(* CODESYS project SHSNU_monitor.project

Project tree, tasks and I/O mapping:
  Device : OWEN PLC323.03-CS.WEB, Owen, order no. 005, version 3.5.0.40
      unmapped channels: Discrete Outputs, Discrete inputs
    application Application
      libraries: CoDeSys Container Library Template, 3.5.3.0 (3S - Smart Software Solutions GmbH); МВА АСКИР, 1.0.0.0 (ООО ПЛАДА); ModBus, 3.1.1 (OWEN); SysCom, 3.5.5.0 (System); ModulsOwenLib, 3.5.4.2 (Production association OWEN); OwenArchiverErrors, 3.5.4.2 (Production association OWEN); CAA Async Manager Extern, * (CAA Technical Workgroup); ArchivatorOwenLib, 3.5.4.2 (OWEN); SysTime23, 3.5.2.0 (System); SysTimeRtc, 3.5.5.0 (System); CAA DTUtil Extern, * (CAA Technical Workgroup); CAA File, 3.5.11.0 (CAA Technical Workgroup); SysSocket, 3.5.9.0 (System); OwenModemLib, 3.5.2.13 (OWEN); BASIC, 3.31 (OSCAT)
      task MainTask (cyclic, interval t#20ms, priority 1, watchdog t#5000ms x 1) calls PLC_PRG
      program PLC_PRG [CFC]
      Symbols
      global variables GVL
      data type Massive
      Code/
        Dop_modules/
          program convert [ST]
          function Duo_Word_to_Real [CFC]
          function block Real_to_Duo_Word [CFC]
          function block Perecl_Perem [ST]
          function block Timer_impuls [CFC]
          function block Schetchik [ST]
          function block NotNull [ST]
          function block IVD3_input_old [ST]
          function block IVD3_input_reg [ST]
          function POU [CFC]
          function block AddInMassive [ST]
          function block IVD3_input [ST]
          function block Auton_val [ST]
        Modules/
          function block DTime [ST]
          function block SPLIT_DT_TO_FSTRINGS [ST]
          function CONCAT11 [ST]
          function LEAD_ZERO [ST]
          function block SMS [CFC]
        Modules_dinamogramma/
          function block MassivCollect [ST]
          function block Create_Shablon [ST]
          function block Alarm_Control [ST]
          function block Correct_Shablon [ST]
          function block Auton_dynamogram_modbus [ST]
          function block Create_Shablon_v2 [ST]
        Modules_parameter/
          function block Calculate_Parameter_Usilie [ST]
          function block Emulate_Parameter_Power [ST]
      data type AlarmLog
    Ethernet : Ethernet, 3S - Smart Software Solutions GmbH, version 3.4.2.0
      ModbusTCP_Slave_Device : ModbusTCP Slave Device, 3S - Smart Software Solutions GmbH, version 3.4.1.10
          settings: Unit-ID = 159
          input  p13 : WORD  // IW0
          input  p14 : WORD  // IW1
          input  p15 : WORD  // IW2
          input  p16 : WORD  // IW3
          input  p17 : WORD  // IW4
          input  p18 : WORD  // IW5
          input  p19 : WORD  // IW6
          input  p20 : WORD  // IW7
          input  p21 : WORD  // IW8
          input  p22 : WORD  // IW9
          unmapped channels: QW0, QW1, QW2, QW3, QW4, QW5, QW6, QW7, QW8, QW9
    Owen:Internal
        output Application.ledError : BOOL  // Discrete Outputs.RELE1
        output Application.ledError : BOOL  // Discrete Outputs.LED_ERROR
        unmapped channels: Discrete Outputs, Discrete inputs
  text list GlobalTextList
  5ce3da45-db07-42e7-a21c-a00fff4ed8f6|D:\Work\Gorizont REP\code\src\Askir\DesktopApp\res\dashboard.jpg
  5ce3da45-db07-42e7-a21c-a00fff4ed8f6|F:\Other\YandexDisk\OVEN\Документация\dashboard.jpg
  5ce3da45-db07-42e7-a21c-a00fff4ed8f6|F:\Other\YandexDisk\OVEN\Проекты\Askir\Askir_materials\Askir_bg.jpg
  5ce3da45-db07-42e7-a21c-a00fff4ed8f6|F:\Other\YandexDisk\OVEN\Проекты\Askir\Askir_materials\ZadPodElDv.jpg
  5ce3da45-db07-42e7-a21c-a00fff4ed8f6|F:\Other\YandexDisk\OVEN\Проекты\Askir\Askir_materials\Askir_bg_lable.jpg
*)

// Device/Application/Massive
TYPE Massive :
STRUCT
	Date_Time: STRING(20);
	var1, var2, var3, var4, var5, var6 : REAL;
END_STRUCT
END_TYPE

// Device/Application/AlarmLog
TYPE AlarmLog :
STRUCT
	Date_Time: STRING(20);
	ShablonIndex:INT;
	ShablonValue:REAL;
	Value:REAL;
	Otklonenie:REAL;
END_STRUCT
END_TYPE

// Device/Application/GVL
VAR_GLOBAL
	var2: REAL;
	
	p1, p2, p3, p4, p5, p6, p7, p8, p9, p10: WORD;
	
	
	VibrA1, VibrA2, VibrA3, VibrB1, VibrB2, VibrB3, VibrC1, VibrC2, VibrC3, VibrD1, VibrD2, VibrD3: REAL;
	(*Вибрация позиция A плоскость X*)		VibrAX:REAL;
	(*Вибрация позиция A плоскость Y*)		VibrAY:REAL;
	(*Вибрация позиция A плоскость Z*)		VibrAZ:REAL;
	
	(*Вибрация позиция B плоскость X*)		VibrBX:REAL;
	(*Вибрация позиция B плоскость Y*)		VibrBY:REAL;
	(*Вибрация позиция B плоскость Z*)		VibrBZ:REAL;
	
	(*Вибрация позиция C плоскость X*)		VibrCX:REAL;
	(*Вибрация позиция C плоскость Y*)		VibrCY:REAL;
	(*Вибрация позиция C плоскость Z*)		VibrCZ:REAL;
	
	(*Динамограмма с датчика усилия*)		Dinamogram: ARRAY[1..Dynamogram_length] OF INT;
	minMnoj: REAL := 0.001;
	maxMnoj: REAL := 100;
	
	minSmesh: REAL := -100;
	maxSmesh: REAL := 100;
	
	Start: BOOL := FALSE;
	
	arrey1111 : ARRAY [1..5] OF INT := [1 , 2, 3, 4, 5];
	ledError: BOOL:=TRUE;
	
	
END_VAR

VAR_GLOBAL RETAIN
	M1, M2, M3, M4, M5, M6, M7, M8, M9, M10, M11, M12: REAL := 1;
	S1, S2, S3, S4, S5, S6, S7, S8, S9, S10, S11, S12: REAL := 0;
	MemM1, MemM2, MemM3, MemM4, MemM5, MemM6, MemM7, MemM8, MemM9, MemM10, MemM11, MemM12: REAL;
	MemS1, MemS2, MemS3, MemS4, MemS5, MemS6, MemS7, MemS8, MemS9, MemS10, MemS11, MemS12: REAL;
	SaveConfig: BOOL;
	
END_VAR

VAR_GLOBAL CONSTANT
	m_MAX_arr: INT:=500; //размер массива	
	Dynamogram_length: INT:=500;
END_VAR

// Device/Application/PLC_PRG
PROGRAM PLC_PRG
VAR
	tp1: TP;
	ErrMDVV: WORD;
	v4: REAL;
	v3: REAL;
	v2: REAL;
	v1: REAL;
	x: BYTE;
	R1, R2, R3, R4, R5, R6, R7, R8, R9, R10, R11, R12, R13, R14, R15, R16, R17, R18, R19, R20, R21, R22: REAL;
	peremR: REAL;
	x3: WORD;
	Perecluchatel: Perecl_Perem;
	RS_0: RS;
	v1_2: REAL;
	v1_3: REAL;
	v2_2: REAL;
	v3_2: REAL;
	v4_2: REAL;
	v1_2IS: WORD;
	v2_2IS: WORD;
	v3_2IS: WORD;
	v4_2IS: WORD;
	v5_2: REAL;
	v6_2: REAL;
	v7_2: REAL;
	v5_2IS: WORD;
	v6_2IS: WORD;
	v7_2IS: WORD;
	v8_2: REAL;
	cicle: WORD;
	Sch_1: Schetchik;
	
	NotNull_1: NotNull;
	NotNull_2: NotNull;
	NotNull_3: NotNull;
	NotNull_4: NotNull;
	NotNull_5: NotNull;
	NotNull_6: NotNull;
	NotNull_7: NotNull;
	NotNull_8: NotNull;
	NotNull_9: NotNull;
	NotNull_10: NotNull;
	
	MConf1,MConf2,MConf3,MConf4,MConf5,MConf6,MConf7,MConf8,MConf9,MConf10,MConf11,MConf12, MConfigTest:REAL := 1;
	SConf1,SConf2,SConf3,SConf4,SConf5,SConf6,SConf7,SConf8,SConf9,SConf10,SConf11,SConf12, SConfigTest:REAL := 1;
	
	
	//IVD3_input_reg_0: IVD3_input_reg;
	//IVD3_input_reg_1: IVD3_input_reg;
	//IVD3_input_reg_2: IVD3_input_reg;
	//IVD3_input_reg_3: IVD3_input_reg;
	
	Port_5: ComConn;
	MV110_8A: MV110_8A_inputs;
	
	MV110_8A_inp_1,
	MV110_8A_inp_2, 
	MV110_8A_inp_3, 
	MV110_8A_inp_4, 
	MV110_8A_inp_5, 
	MV110_8A_inp_6, 
	MV110_8A_inp_7, 
	MV110_8A_inp_8: REAL;
	
	ComConn_Tablo: ComConn;
	Write_in_Tablo: UniWrite;
	ComConn_Vibro: ComConn;
	SR_0: RS;
	

	


	DTime_0: DTime;
	
	systimestring:string;
	vcb: DWORD;

	
	testMassiv: Massive := (Date_Time:= systimestring, var1:=VibrAZ, var2:=VibrAX, var3:=VibrAY, var4:=VibrBZ, var5:=VibrBX, var6:=VibrBY);
	AddInMassive_0: AddInMassive;
	
	
	MassivIVD3_1, MassivIVD3_2, MassivIVD3_3: ARRAY [0..gvl.m_MAX_arr] OF REAL;
	timeMassiveIVD3_1, timeMassiveIVD3_2, timeMassiveIVD3_3: STRING;
	
	TP_add_massiv: TP;
	RS_TP: RS;
	Emulate_Parameter_Power_test: Emulate_Parameter_Power;
	
	Power_U: REAL;
	Power_I: REAL;
	Power_Work_Hod:REAL;
	Power_Work_Up:REAL;
	Power_Work_Down:REAL;
	Power_Min:REAL;
	Power_Max:REAL;
	Power_Razmah:REAL;
	
	Calculate_Parameter_Usilie_0: Calculate_Parameter_Usilie;
	
	Usilie_Work_Hod:REAL;
	Usilie_Work_Up:REAL;
	Usilie_Work_Down:REAL;
	Usilie_Raznica:REAL;
	Usilie_Min:REAL;
	Usilie_Max:REAL;
	Usilie_Razmah:REAL;
	ComConn_Sim: comconn;
	modem_fb: FB_SMS_CSD;
	
	newSMS, newRing, CSD, modem_busy: BOOL;
	
	tesTP: bool;
	TON_0, TON_1, TON_2: ton;
	start: bool := true;
	R_TRIG_0: R_TRIG;
	F_TRIG_0: F_TRIG;
	TON_3: ton;
	RS_1: rs;
	qwe: IVD3_input_reg;
	asd: IVD3_input_reg;
	zxc: IVD3_input_reg;
	IVD3_input_reg_0: IVD3_input_reg;
	Auton_val_0: Auton_val;
	auton_value: INT;
	MassivCollect_Dynamogram: MassivCollect;
	masDynamogram: ARRAY [0..gvl.m_MAX_arr] OF REAL;
	timeDynamogram: STRING;
	auton_val_time: STRING;
	TP_work: TP;
	Start_work: BOOL:= false;
	IVD3_A: IVD3_input_reg;
	IVD3_B: IVD3_input_reg;
	IVD3_C: IVD3_input_reg;
END_VAR
VAR // added by the converter: edge detectors and wires of the graphical bodies
    _w1 : BYTE;
END_VAR

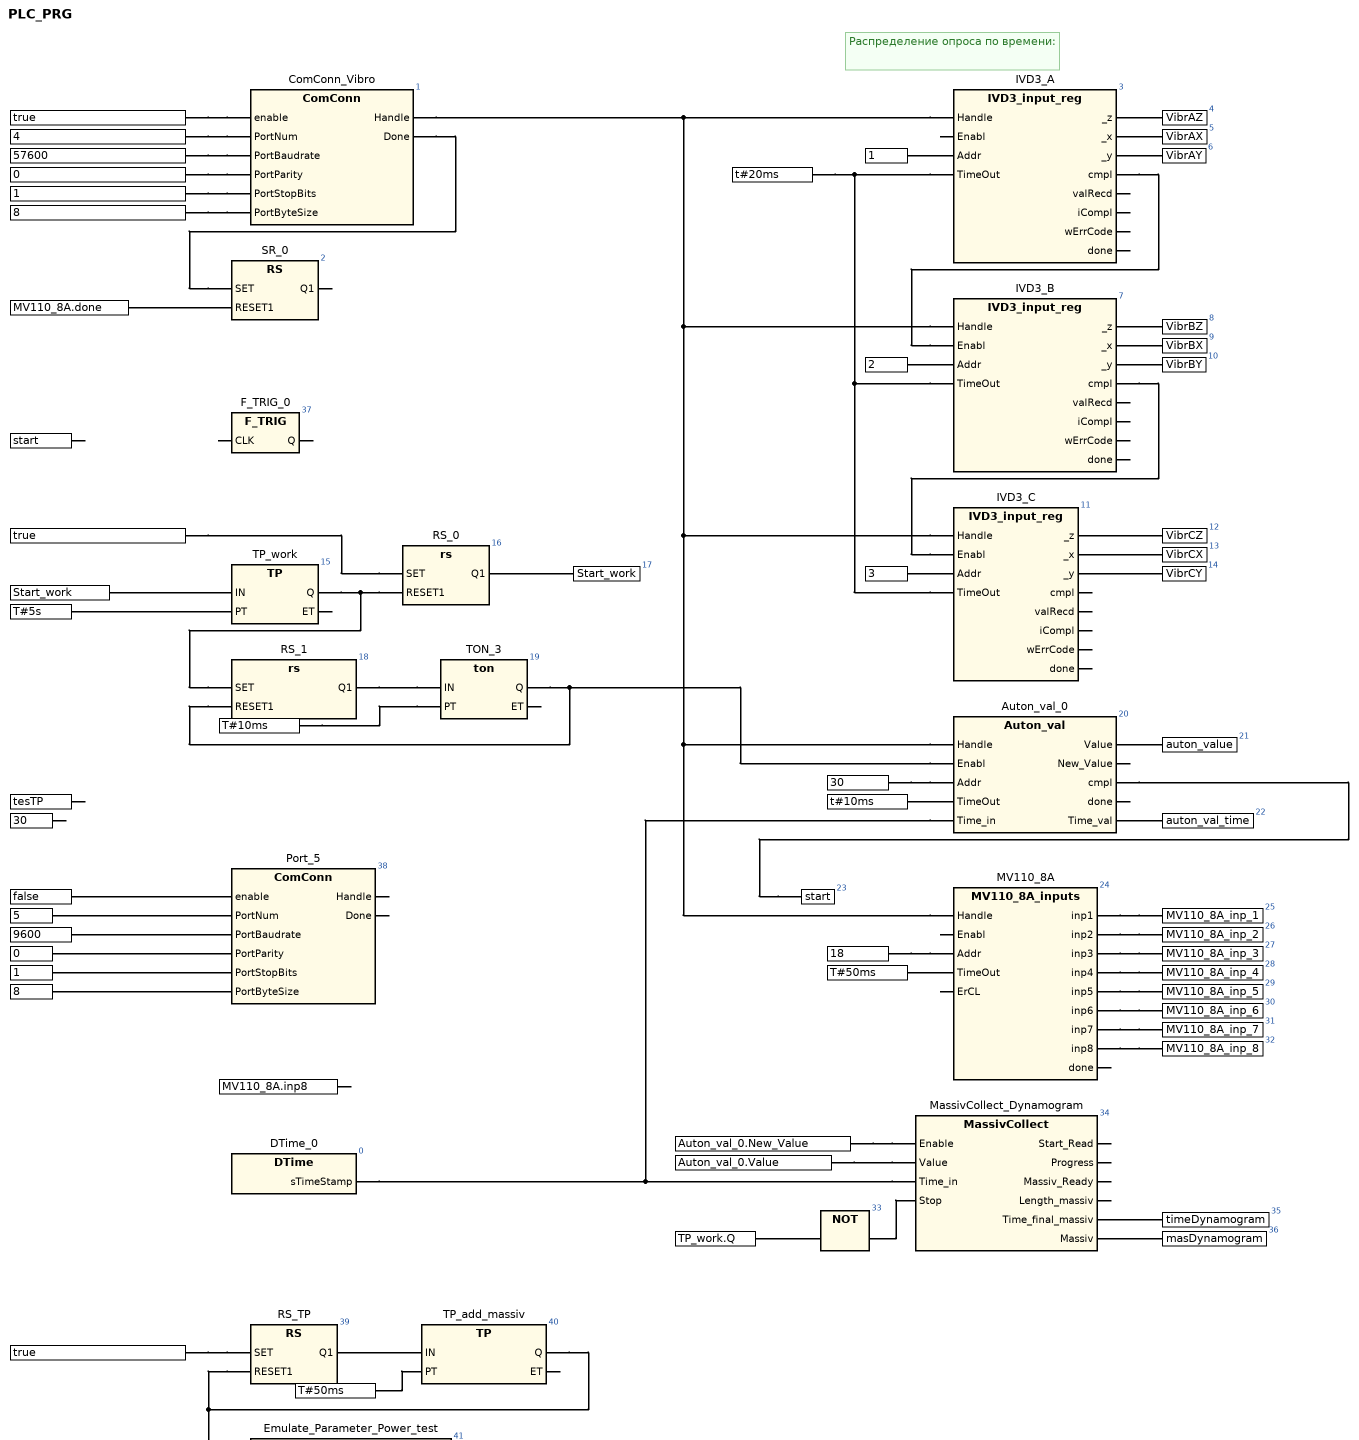
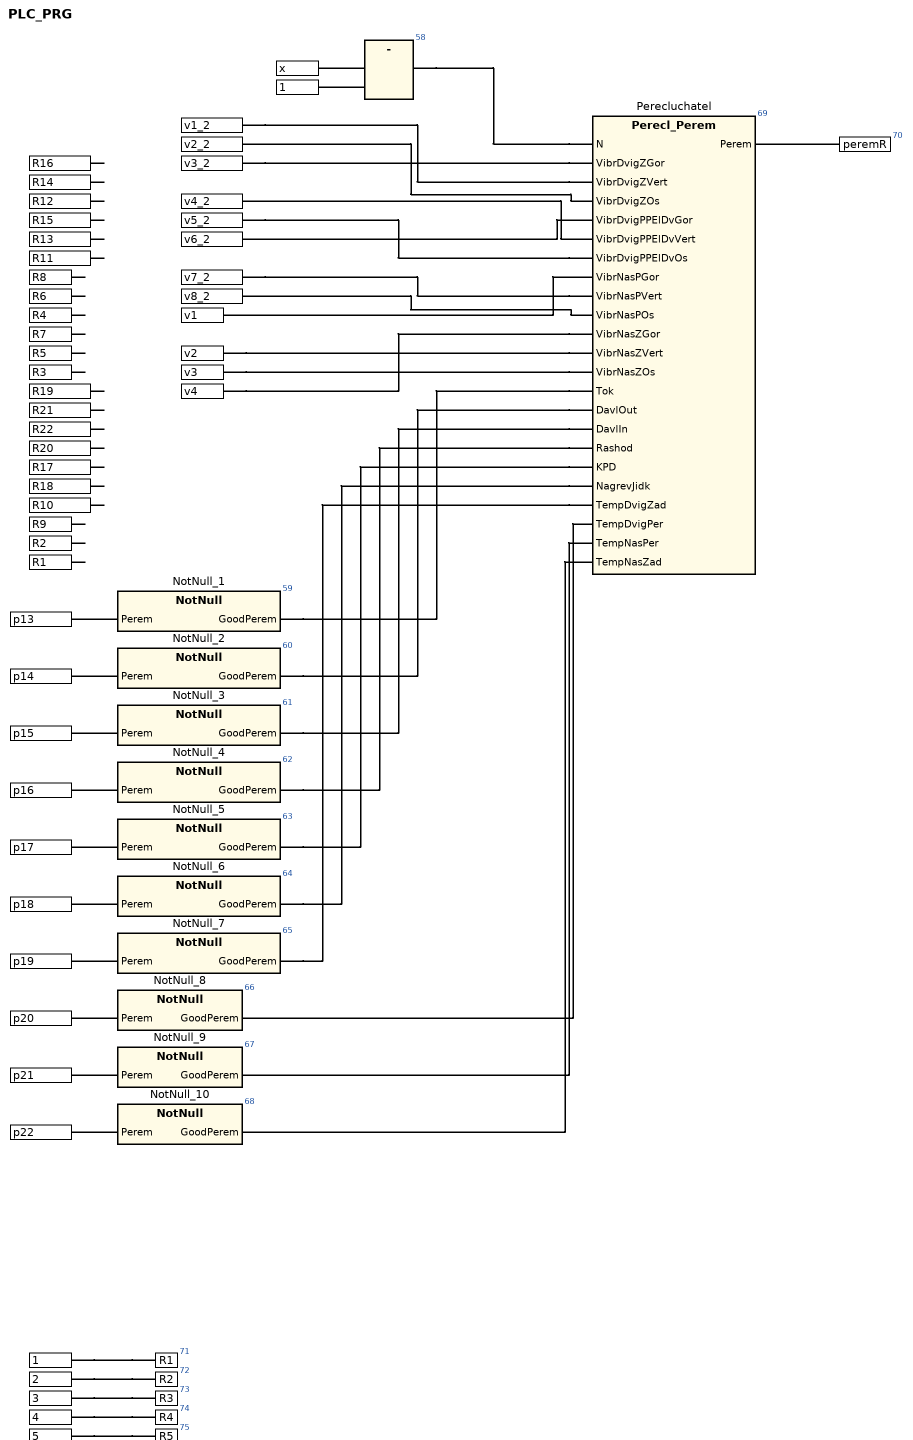
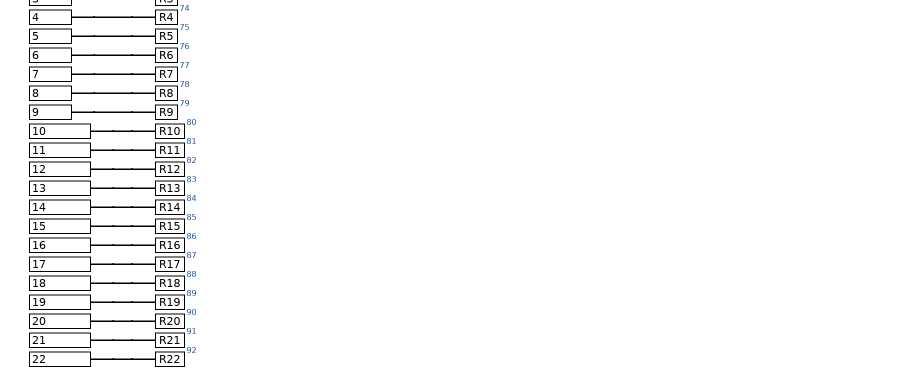
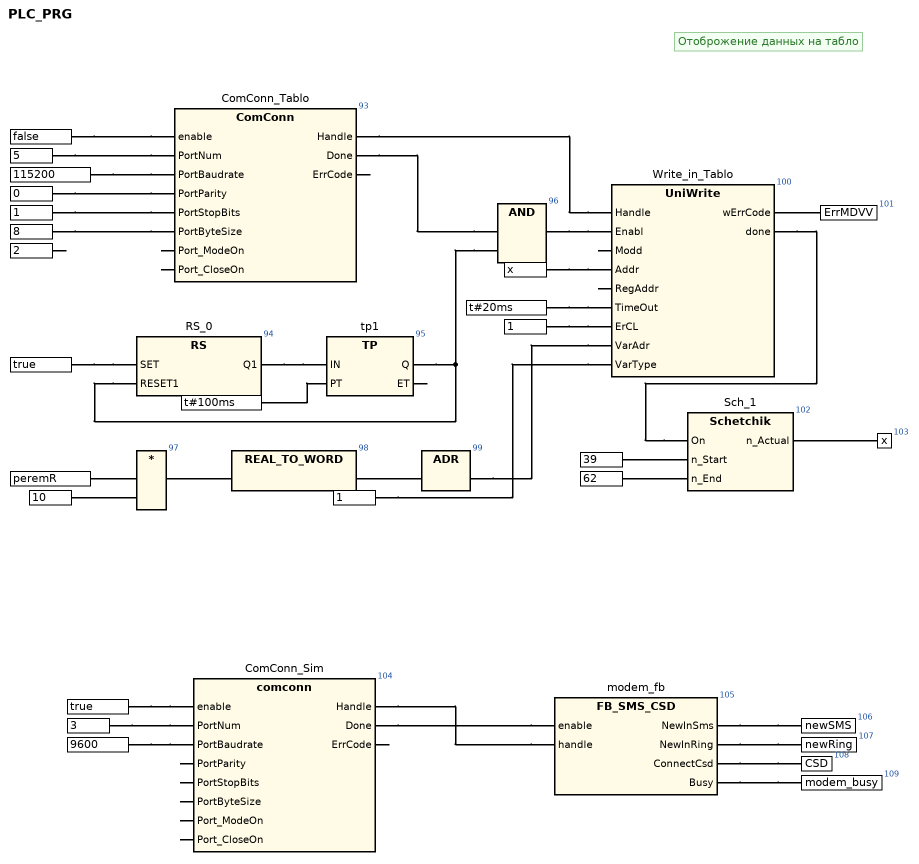
DTime_0(); // DTime
ComConn_Vibro(
    enable := true,
    PortNum := 4,
    PortBaudrate := 57600,
    PortParity := 0,
    PortStopBits := 1,
    PortByteSize := 8); // ComConn
SR_0(SET := ComConn_Vibro.Done, RESET1 := MV110_8A.done); // RS
// Распределение опроса по времени:
IVD3_A(Handle := ComConn_Vibro.Handle, Addr := 1, TimeOut := t#20ms); // IVD3_input_reg
VibrAZ := IVD3_A._z;
VibrAX := IVD3_A._x;
VibrAY := IVD3_A._y;
IVD3_B(Handle := ComConn_Vibro.Handle, Enabl := IVD3_A.cmpl, Addr := 2, TimeOut := t#20ms); // IVD3_input_reg
VibrBZ := IVD3_B._z;
VibrBX := IVD3_B._x;
VibrBY := IVD3_B._y;
IVD3_C(Handle := ComConn_Vibro.Handle, Enabl := IVD3_B.cmpl, Addr := 3, TimeOut := t#20ms); // IVD3_input_reg
VibrCZ := IVD3_C._z;
VibrCX := IVD3_C._x;
VibrCY := IVD3_C._y;
TP_work(IN := Start_work, PT := T#5s); // TP
RS_0(SET := true, RESET1 := TP_work.Q); // rs
Start_work := RS_0.Q1;
RS_1(SET := TP_work.Q, RESET1 := TON_3.Q); // rs
TON_3(IN := RS_1.Q1, PT := T#10ms); // ton
Auton_val_0(
    Handle := ComConn_Vibro.Handle,
    Enabl := TON_3.Q,
    Addr := 30,
    TimeOut := t#10ms,
    Time_in := DTime_0.sTimeStamp); // Auton_val
auton_value := Auton_val_0.Value;
auton_val_time := Auton_val_0.Time_val;
start := Auton_val_0.cmpl;
MV110_8A(Handle := ComConn_Vibro.Handle, Addr := 18, TimeOut := T#50ms); // MV110_8A_inputs
MV110_8A_inp_1 := MV110_8A.inp1;
MV110_8A_inp_2 := MV110_8A.inp2;
MV110_8A_inp_3 := MV110_8A.inp3;
MV110_8A_inp_4 := MV110_8A.inp4;
MV110_8A_inp_5 := MV110_8A.inp5;
MV110_8A_inp_6 := MV110_8A.inp6;
MV110_8A_inp_7 := MV110_8A.inp7;
MV110_8A_inp_8 := MV110_8A.inp8;
MassivCollect_Dynamogram(
    Enable := Auton_val_0.New_Value,
    Value := Auton_val_0.Value,
    Time_in := DTime_0.sTimeStamp,
    Stop := NOT TP_work.Q); // MassivCollect
timeDynamogram := MassivCollect_Dynamogram.Time_final_massiv;
masDynamogram := MassivCollect_Dynamogram.Massiv;
F_TRIG_0(); // F_TRIG
Port_5(
    enable := false,
    PortNum := 5,
    PortBaudrate := 9600,
    PortParity := 0,
    PortStopBits := 1,
    PortByteSize := 8); // ComConn
RS_TP(SET := true, RESET1 := TP_add_massiv.Q); // RS
TP_add_massiv(IN := RS_TP.Q1, PT := T#50ms); // TP
Emulate_Parameter_Power_test(
    Enable := TP_add_massiv.Q,
    U_Random_Min := 370,
    U_Random_Max := 390,
    I_Random_Min := 40,
    I_Random_Max := 60,
    Index := MassivCollect_Dynamogram.Progress); // Emulate_Parameter_Power
Power_U := Emulate_Parameter_Power_test.U;
Power_I := Emulate_Parameter_Power_test.I;
Power_Work_Up := Emulate_Parameter_Power_test.Work_Up;
Power_Work_Down := Emulate_Parameter_Power_test.Work_Down;
Power_Work_Hod := Emulate_Parameter_Power_test.Work_Hod;
Power_Max := Emulate_Parameter_Power_test.Max_Power;
Power_Min := Emulate_Parameter_Power_test.Min_Power;
Power_Razmah := Emulate_Parameter_Power_test.Razmah;
Calculate_Parameter_Usilie_0(
    Enable := MassivCollect_Dynamogram.Massiv_Ready,
    Index := MassivCollect_Dynamogram.Progress,
    Dinamogramma := MassivCollect_Dynamogram.Massiv); // Calculate_Parameter_Usilie
Usilie_Work_Up := Calculate_Parameter_Usilie_0.Work_Up;
Usilie_Work_Down := Calculate_Parameter_Usilie_0.Work_Down;
Usilie_Work_Hod := Calculate_Parameter_Usilie_0.Work_Hod;
Usilie_Raznica := Calculate_Parameter_Usilie_0.Raznica;
Usilie_Max := Calculate_Parameter_Usilie_0.Max_Usil;
Usilie_Min := Calculate_Parameter_Usilie_0.Min_Usil;
Usilie_Razmah := Calculate_Parameter_Usilie_0.Razmah;
_w1 := x - 1;
NotNull_1(Perem := p13); // NotNull
NotNull_2(Perem := p14); // NotNull
NotNull_3(Perem := p15); // NotNull
NotNull_4(Perem := p16); // NotNull
NotNull_5(Perem := p17); // NotNull
NotNull_6(Perem := p18); // NotNull
NotNull_7(Perem := p19); // NotNull
NotNull_8(Perem := p20); // NotNull
NotNull_9(Perem := p21); // NotNull
NotNull_10(Perem := p22); // NotNull
Perecluchatel(
    N := _w1,
    VibrDvigZGor := v3_2,
    VibrDvigZVert := v1_2,
    VibrDvigZOs := v2_2,
    VibrDvigPPElDvGor := v6_2,
    VibrDvigPPElDvVert := v4_2,
    VibrDvigPPElDvOs := v5_2,
    VibrNasPGor := v1,
    VibrNasPVert := v7_2,
    VibrNasPOs := v8_2,
    VibrNasZGor := v4,
    VibrNasZVert := v2,
    VibrNasZOs := v3,
    Tok := NotNull_1.GoodPerem,
    DavlOut := NotNull_2.GoodPerem,
    DavlIn := NotNull_3.GoodPerem,
    Rashod := NotNull_4.GoodPerem,
    KPD := NotNull_5.GoodPerem,
    NagrevJidk := NotNull_6.GoodPerem,
    TempDvigZad := NotNull_7.GoodPerem,
    TempDvigPer := NotNull_8.GoodPerem,
    TempNasPer := NotNull_9.GoodPerem,
    TempNasZad := NotNull_10.GoodPerem); // Perecl_Perem
peremR := Perecluchatel.Perem;
R1 := 1;
R2 := 2;
R3 := 3;
R4 := 4;
R5 := 5;
R6 := 6;
R7 := 7;
R8 := 8;
R9 := 9;
R10 := 10;
R11 := 11;
R12 := 12;
R13 := 13;
R14 := 14;
R15 := 15;
R16 := 16;
R17 := 17;
R18 := 18;
R19 := 19;
R20 := 20;
R21 := 21;
R22 := 22;
ComConn_Tablo(
    enable := false,
    PortNum := 5,
    PortBaudrate := 115200,
    PortParity := 0,
    PortStopBits := 1,
    PortByteSize := 8); // ComConn
RS_0(SET := true, RESET1 := tp1.Q); // RS
tp1(IN := RS_0.Q1, PT := t#100ms); // TP
// Отоброжение данных на табло
Write_in_Tablo(
    Handle := ComConn_Tablo.Handle,
    Enabl := ComConn_Tablo.Done AND tp1.Q,
    Addr := x,
    TimeOut := t#20ms,
    ErCL := 1,
    VarAdr := ADR(REAL_TO_WORD(peremR * 10)),
    VarType := 1); // UniWrite
ErrMDVV := Write_in_Tablo.wErrCode;
Sch_1(On := Write_in_Tablo.done, n_Start := 39, n_End := 62); // Schetchik
x := Sch_1.n_Actual;
ComConn_Sim(enable := true, PortNum := 3, PortBaudrate := 9600); // comconn
modem_fb(enable := ComConn_Sim.Done, handle := ComConn_Sim.Handle); // FB_SMS_CSD
newSMS := modem_fb.NewInSms;
newRing := modem_fb.NewInRing;
CSD := modem_fb.ConnectCsd;
modem_busy := modem_fb.Busy;
// start: input not connected
// tesTP: input not connected
// 30: input not connected
// MV110_8A.inp8: input not connected
// MassivCollect_Dynamogram.Length_massiv: input not connected
// R16: input not connected
// R14: input not connected
// R12: input not connected
// R15: input not connected
// R13: input not connected
// R11: input not connected
// R8: input not connected
// R6: input not connected
// R4: input not connected
// R7: input not connected
// R5: input not connected
// R3: input not connected
// R19: input not connected
// R21: input not connected
// R22: input not connected
// R20: input not connected
// R17: input not connected
// R18: input not connected
// R10: input not connected
// R9: input not connected
// R2: input not connected
// R1: input not connected
// 2: input not connected

END_PROGRAM

// Device/Application/Code/Modules/DTime
FUNCTION_BLOCK DTime
VAR_OUTPUT
	sTimeStamp:						STRING(20);							// метка времени в виде форматированной строки
END_VAR
VAR
	fbGetCurrentDT:					DTU.GetDateAndTime;					// ФБ считывания системного времени	
	fbSplitDT:						SPLIT_DT_TO_FSTRINGS;				// ФБ конвертации времени в строку
	asDateTimeStrings:				ARRAY [0..10] OF STRING;			// метка времени в виде отдельных строковых разрядов
	
END_VAR
VAR CONSTANT
	// заголовок архива
	c_sTitle:						STRING(60)	:=	'Дата;Время;Значение типа WORD;Значение типа REAL;$N';
	c_sDelimiter:					STRING(1)	:=	';';
END_VAR

// считываем системное время
fbGetCurrentDT(xExecute:=NOT(fbGetCurrentDT.xDone));

IF fbGetCurrentDT.xDone THEN
	// вырезаем отдельные разряды времени и конвертируем их в строки
	fbSplitDT(dtDateAndTime:=fbGetCurrentDT.dtDateAndTime);
END_IF

// подготавливаем метку времени в виде форматированной строки
asDateTimeStrings[0]	:=	fbSplitDT.sDay;
asDateTimeStrings[1]	:=	'.';
asDateTimeStrings[2]	:=	fbSplitDT.sMonth;
asDateTimeStrings[3]	:=	'.';
asDateTimeStrings[4]	:=	fbSplitDT.sYear;
asDateTimeStrings[5]	:=	c_sDelimiter;
asDateTimeStrings[6]	:=	fbSplitDT.sHour;
asDateTimeStrings[7]	:=	':';
asDateTimeStrings[8]	:=	fbSplitDT.sMinute;
asDateTimeStrings[9]	:=	':';
asDateTimeStrings[10]	:=	fbSplitDT.sSecond;

// собираем дату и время в строку
sTimeStamp:= CONCAT11(asDateTimeStrings);

END_FUNCTION_BLOCK

// Device/Application/Code/Modules/CONCAT11
// функция склеивает заданное число строковых переменных, помещенных в массив

FUNCTION CONCAT11 : STRING(255)
VAR_INPUT
	asSTR:			ARRAY [0..c_MAX_STR] OF STRING;
END_VAR
VAR
	sBuffer:		STRING;			// промежуточная переменная
	i:				INT;			// счетчик для цикла
END_VAR

VAR CONSTANT
	c_MAX_STR:		INT:=10;		// размер массива строковых переменных
END_VAR

FOR i:=0 TO c_MAX_STR DO
	sBuffer:=CONCAT(sBuffer, asSTR[i]);
END_FOR

CONCAT11:=sBuffer;

END_FUNCTION

// Device/Application/Code/Modules/SPLIT_DT_TO_FSTRINGS
// ФБ разделяет метку времени типа DT на строковые представления отдельных разрядов с ведущими нулями

FUNCTION_BLOCK SPLIT_DT_TO_FSTRINGS
VAR_INPUT
	dtDateAndTime:			DT;			// метка времени в формате DT
END_VAR
VAR_OUTPUT
	sYear:					STRING;		// разряды времени в строковом представлении
	sMonth:					STRING;		//
	sDay:					STRING;		//
	sHour:					STRING;		//
	sMinute:				STRING;		//
	sSecond:				STRING;		//
END_VAR
VAR
	uiYear:					UINT;		// разряды времени в десятичном представлении
	uiMonth:				UINT;		//
	uiDay:					UINT;		//
	uiHour:					UINT;		//
	uiMinute:				UINT;		//
	uiSecond:				UINT;		//
END_VAR

DTU.DTSplit
(
	dtDateAndTime,
	ADR(uiYear),
	ADR(uiMonth),
	ADR(uiDay),
	ADR(uiHour),
	ADR(uiMinute),
	ADR(uiSecond)
);

sYear		:=		UINT_TO_STRING(uiYear);
sMonth		:=		LEAD_ZERO(uiMonth);
sDay		:=		LEAD_ZERO(uiDay);
sHour		:=		LEAD_ZERO(uiHour);
sMinute		:=		LEAD_ZERO(uiMinute);
sSecond		:=		LEAD_ZERO(uiSecond);

END_FUNCTION_BLOCK

// Device/Application/Code/Modules/LEAD_ZERO
// функция преобразует число в строку с ведущим нулем

FUNCTION LEAD_ZERO : STRING
VAR_INPUT
	uiInput:		 UINT;
END_VAR
VAR
END_VAR

IF uiInput>9 THEN
	LEAD_ZERO:=UINT_TO_STRING(uiInput);
ELSE 
	LEAD_ZERO:=CONCAT('0', UINT_TO_STRING(uiInput));
END_IF

END_FUNCTION

// Device/Application/Code/Dop_modules/IVD3_input_reg
FUNCTION_BLOCK IVD3_input_reg
VAR_INPUT
	(*идентификатор порта*)											Handle:SysCom.RTS_IEC_HANDLE;
	(*разрешение на работу*)											Enabl:BOOL;
	(*адресс прибора, по умолчанию 1*)						Addr:BYTE:=1;
	(*таймаут, по умолчанию 30мс*)								TimeOut: TIME:=T#30MS;
	
	

END_VAR
VAR_OUTPUT
	(*измеренное значение плоскости Z*)			_z:REAL;
	(*измеренное значение плоскости X*)			_x:REAL;
	(*измеренное значение плоскости Y*)			_y:REAL;
	
	cmpl:BOOL;
	valRecd:bool;
	iCompl:UINT;
	(*код ошибки*)										wErrCode:WORD;
	(*флаг завершения*)									done:BOOL;
END_VAR
VAR
	(*режим работы ModBus (MB_RTU, MB_Ascii), по умолчанию RTU*)	Modd:MB_MODE:=MB_RTU ;
	(*адресс регистра, по умолчанию 0*)								RegAddr:WORD:=16#0;
	(*число перезапросов, по умолчанию 3*)							ErCL:BYTE:=3;
	ErrCount:BYTE:=0;
	
	shag:byte:=0;
	err:WORD;
	Exception: BYTE;
	DataSize: WORD;
	KolReg:BYTE;
	get_modbus:MB_RD_INP_REGS;
	//get_modbus2:MB_RD_INP_REGS;
	BUFFER: ARRAY [0..255] OF BYTE;
	i: WORD;
	
	x, y, z: REAL;
	ptr_x, ptr_y, ptr_z:POINTER TO BYTE;
	
	rtrig:R_TRIG;
	trig:rs;
END_VAR

done:=FALSE;
valRecd:=FALSE;

rtrig(clk:=(Enabl));
trig(set:=rtrig.Q,RESET1:=FALSE);


get_modbus(
	Enable:=trig.Q1 ,			(* разрешение работы блока *)
	Mode:=Modd ,		(*режим передачи*)
	DevAddr:=Addr ,			(*адрес*)
	FirstAddr:=RegAddr ,			(*номер регистра*)
	Quantity:=6,			(*количество регистров*)
	ComHandle:=handle ,(*номер COM-порта*)
	TimeOut:=TimeOut , 		(*Таймаут T#30ms*)
	Buffer:=Buffer ,		(* буфер данных *)
	Complete=>cmpl ,		(* скопировать признак завершения операции *)
	Exception=>Err ,		(* скопировать регистр ошибок *)
	ByteCnt=>DataSize );		(*кол-во считанных байтов *)

//IF cmpl=TRUE THEN
//	IF iCompl>=65500 THEN
//		iCompl:=0;
//	END_IF
//	iCompl:=iCompl+1;
//END_IF


	//IF cmpl THEN
		IF Err=0 THEN	
			IF DataSize=17 THEN
//cmpl:=FALSE;
		z:=0;
		ptr_z:=ADR(z);
		ptr_z^:=buffer[4];
		ptr_z:=ptr_z+1;
		ptr_z^:=buffer[3];
		ptr_z:=ptr_z+1;
		ptr_z^:=buffer[6];
		ptr_z:=ptr_z+1;
		ptr_z^:=buffer[5];
		_z:=z;
		
		x:=0;
		ptr_x:=ADR(x);
		ptr_x^:=buffer[8];
		ptr_x:=ptr_x+1;
		ptr_x^:=buffer[7];
		ptr_x:=ptr_x+1;
		ptr_x^:=buffer[10];
		ptr_x:=ptr_x+1;
		ptr_x^:=buffer[9];
		_x:=x;
		
		y:=0;
		ptr_y:=ADR(y);
		ptr_y^:=buffer[12];
		ptr_y:=ptr_y+1;
		ptr_y^:=buffer[11];
		ptr_y:=ptr_y+1;
		ptr_y^:=buffer[14];
		ptr_y:=ptr_y+1;
		ptr_y^:=buffer[13];
		_y:=y;
			
		valRecd:= true;

		done:=TRUE;
		trig(RESET1:=TRUE);
		ErrCount:=0;
		wErrCode:=Err;
		IF iCompl>=65500 THEN
			iCompl:=0;
		END_IF
	iCompl:=iCompl+1;
	ELSE
	ErrCount:=ErrCount+1;
		IF (ErrCount >= ErCL) THEN
			ErrCount:=0;
			done:=TRUE;
			trig(RESET1:=TRUE);
			wErrCode:=Err;
		END_IF
	END_IF
END_IF

//END_IF

END_FUNCTION_BLOCK

// Device/Application/Code/Dop_modules/Auton_val
FUNCTION_BLOCK Auton_val
VAR_INPUT
	(*идентификатор порта*)													Handle:SysCom.RTS_IEC_HANDLE;
	(*разрешение на работу*)													Enabl:BOOL;
	(*адресс прибора, по умолчанию 1*)								Addr:BYTE:=30;
	(*таймаут, по умолчанию 30мс*)										TimeOut: TIME:=T#20MS;
	(*на выходе получим время переменной*)						Time_in: STRING;
END_VAR
VAR_OUTPUT
	(*Собранное значение*) 													Value:INT;
	(*Изменение знасения*)													New_Value:BOOL;
	(*Статус получения ответа после запроса*)					cmpl:BOOL;
	(*флаг завершения*)															done: BOOL;
	(*Время создания переменной*) 										Time_val: STRING;
END_VAR
VAR
	(*режим работы ModBus (MB_RTU, MB_Ascii)*)						Modd:MB_MODE:=MB_RTU ;
	(*адресс регистра, по умолчанию 0*)								RegAddr:WORD:=16#F0;
	(*число перезапросов, по умолчанию 3*)						ErCL:BYTE:=3;
	(*Объект для общения по протоколу modbus*)					get_modbus:MB_RD_HOLD_REGS;
	(*Буфер для принятых байт ответа*)								BUFFER: ARRAY [0..255] OF BYTE;
	
	(*Количество ошибок*)														ErrCount:BYTE:=0;
	(*Регистр ошибок*)																err:WORD;
	(*Количество считанных байт*)											DataSize: WORD;
	
	(*Значение из ответа*)														_value:INT;
	(*Указатель переменной*) 												ptr_value:POINTER TO BYTE;
	(*Переключатель состояний (true/false) *)							rtrig:R_TRIG;
	(*Переключатель состояний (true/false)*)							RStrig:rs;

END_VAR

done:=FALSE;
New_Value:= FALSE;


rtrig(clk:=(Enabl));
RStrig(set:=rtrig.Q, RESET1:=FALSE);

get_modbus(
	Enable:=RStrig.Q1 ,				(* разрешение работы блока *)
	Mode:=Modd ,					(*режим передачи*)
	DevAddr:=Addr ,				(*адрес*)
	FirstAddr:=RegAddr ,		(*номер регистра*)
	Quantity:=1,						(*количество регистров*)
	ComHandle:=handle ,		(*номер COM-порта*)
	TimeOut:=TimeOut , 		(*Таймаут T#30ms*)
	Buffer:=Buffer ,					(* буфер данных *)
	Complete=>cmpl ,			(* скопировать признак завершения операции *)
	Exception=>Err ,				(* скопировать регистр ошибок *)
	ByteCnt=>DataSize );		(*кол-во считанных байтов *)
	
IF Err=0 THEN	
	IF DataSize=7 THEN
		_value:=0;
		ptr_value:=ADR(_value);
		ptr_value^:=buffer[4];
		ptr_value:=ptr_value+1;
		ptr_value^:=buffer[3];
		Value:=_value;
		Time_val:=Time_in;
		New_Value:=TRUE;
		
		
		//New_Value:= newVal_trig.Q;
		ErrCount:=0;
		done:=TRUE;
		RStrig(RESET1:=TRUE);
		
	ELSE
	ErrCount:=ErrCount+1;
		IF (ErrCount >= ErCL) THEN
			ErrCount:=0;
			done:=TRUE;
			RStrig(RESET1:=TRUE);
			//wErrCode:=Err;
		END_IF
	END_IF
		
END_IF

//Enabl:=FALSE;

END_FUNCTION_BLOCK

// Device/Application/Code/Modules_dinamogramma/MassivCollect
FUNCTION_BLOCK MassivCollect
VAR_INPUT
	Enable : BOOL;
	Value: REAL;
	Time_in: STRING;
	(*Остановить накопление и предоставить*)Stop:BOOL;
END_VAR
VAR_OUTPUT
	Start_Read: BOOL;
	Progress: INT;
	(*Индикатор готовности массива*) Massiv_Ready: BOOL;
	(*Длина массива на момент готовности*) Length_massiv:int;
	(*Время завершения сборки массива*) Time_final_massiv: STRING;
	(*Массив с данными*) Massiv: ARRAY[0..gvl.m_MAX_arr] OF REAL;
END_VAR
VAR
	mBuffer: ARRAY[0..gvl.m_MAX_arr] OF REAL; //промежуточная переменная
	oldBuffer: ARRAY[0..gvl.m_MAX_arr] OF REAL; //промежуточная переменная
	i: INT; //счетчик для цикла
	inWork:BOOL:= FALSE;
	
	createShablon: Create_Shablon_v2;
	createShablonState: BOOL;
	shablon: ARRAY[0..500] OF REAL;
	
	correctShablon: Correct_Shablon;
	alarmControl: Alarm_Control;
	
	firstStop:bool:=true;
END_VAR
VAR CONSTANT
	//m_MAX_arr: INT:=200; //размер массива	
	
END_VAR

IF Enable THEN			
		// если работа окончена сбрасываем все параметры
		IF inWork=FALSE THEN
			Start_Read:=FALSE;
			Massiv_Ready:=FALSE;
			Progress:=0;
			FOR i:=0 TO m_MAX_arr DO
				mBuffer[i]:=0;
			END_FOR
			stop:=FALSE;
		END_IF
		
		
		//createShablon( Prohod:= 5, Value:=Value, Index:= Progress, Size_dinamo:=Length_massiv);
		createShablonState:= createShablon.State;
		IF NOT createShablonState THEN 
			shablon:= createShablon.Shablon;
		END_IF
		
		
		alarmControl(Shablon:=shablon, Value:=Value, Index:=Progress, Otklonenie:=80);
		ledError:=alarmControl.Alarm;
		
		inWork:=TRUE;
		Start_Read:= TRUE;
		mBuffer[Progress]:=Value;
		

		Progress:=Progress+1;
		
		Start_Read:= false;
		
		// проверка наполненности массива
		IF (Progress =  m_MAX_arr+1) OR (Stop) THEN
			Massiv_Ready:=TRUE;
			Time_final_massiv:=Time_in;
			oldBuffer:=Massiv;
			Massiv := mBuffer;
			inWork:= FALSE;
			length_massiv:=Progress;
			
			correctShablon( Enable:= Massiv_Ready, Old_Shablon:=shablon, m_MAX_arr:=length_massiv, New_Dinamo:= Massiv);
			shablon:= correctShablon.Shablon;
		END_IF
		
		Enable:=FALSE;
		firstStop:=true;
END_IF

IF  Stop AND firstStop THEN
	Massiv_Ready:=TRUE;
	Time_final_massiv:=Time_in;
	oldBuffer:=Massiv;
	Massiv := mBuffer;
	inWork:= FALSE;
	length_massiv:=Progress;
	
	correctShablon( Enable:= Massiv_Ready, Old_Shablon:=shablon, m_MAX_arr:=length_massiv, New_Dinamo:= Massiv);
	shablon:= correctShablon.Shablon;
	firstStop:=FALSE;
END_IF
createShablon( Prohod:= 5, Massive:=Massiv, StateMassive:= Massiv_Ready);

END_FUNCTION_BLOCK

// Device/Application/Code/Modules_dinamogramma/Create_Shablon_v2
// Формирование шаблона динамограммы с использованием некоторого количеаства проходов
FUNCTION_BLOCK Create_Shablon_v2
VAR_INPUT
	Prohod: INT;
	Massive: ARRAY[0..500] OF REAL;
	StateMassive: BOOL;
	ResetState:BOOL:=FALSE;
	//Size_dinamo:INT;
END_VAR
VAR_OUTPUT
	State: BOOL;
	Shablon: ARRAY[0..500] OF REAL;
END_VAR
VAR
	
	shablonBufer: ARRAY[0..500] OF REAL;
	prohod_i:INT:=1;
	i:INT;
	ci: INT;
END_VAR

IF ResetState=TRUE THEN
	State:=FALSE;
	ResetState:=false;
END_IF

IF State=FALSE THEN
	// Если количество проходов еще не истекло, то выполняем сбор данных
	IF Prohod >= prohod_i THEN
		IF StateMassive=TRUE THEN
			FOR ci:=0 TO 500 DO
				shablonBufer[ci]:=shablonBufer[ci] + Massive[ci];
			END_FOR
		//shablonBufer:=shablonBufer+Massive;
		prohod_i:= prohod_i + 1;
		END_IF
		
	// Если получены все массивы, делим на кол-во проходов и получаем среднее значение
	IF Prohod = prohod_i THEN
		FOR ci:=0 TO 500 DO
				shablonBufer[ci]:=shablonBufer[ci] /Prohod;
			END_FOR
		//shablonBufer:=shablonBufer/Prohod; // это не работает
			//FOR i:=0 TO Size_dinamo DO
			//	shablonBufer[i]:= shablonBufer[i]/Prohod;
			//END_FOR
			State:= TRUE;	// Выставляем флаг о завершернии в TRUE
			Shablon:= shablonBufer; 	// Предоставляем полученный усредненный массив
		END_IF 
	END_IF
END_IF

END_FUNCTION_BLOCK

// Device/Application/Code/Modules_dinamogramma/Correct_Shablon
// Корректировка существующего шаблона на основании рабочих показаний
FUNCTION_BLOCK Correct_Shablon
VAR_INPUT
	Enable: BOOL;
	Old_Shablon: ARRAY[0..500] OF REAL;
	m_MAX_arr:INT;
	New_Dinamo:ARRAY[0..gvl.m_MAX_arr] OF REAL;
END_VAR
VAR_OUTPUT
	Shablon: ARRAY[0..500] OF REAL;
END_VAR
VAR
	i:INT;
	shablonBufer: ARRAY[0..500] OF REAL;
END_VAR

IF  Enable THEN
	// получив все необходимые данные проходим по массиву
	FOR i:=0 TO m_MAX_arr DO
		//на основе перечня условий формируем новый шаблон
		
		IF Old_Shablon[i]=0 AND New_Dinamo[i]=0 THEN
			shablonBufer[i]:=0;
		END_IF
		
		IF Old_Shablon[i]=0 AND New_Dinamo[i]<>0 THEN
			shablonBufer[i]:=New_Dinamo[i];
		END_IF
	
		IF Old_Shablon[i]<>0 AND New_Dinamo[i]<>0 THEN
			shablonBufer[i]:= (Old_Shablon[i]+New_Dinamo[i])/2;
		END_IF
		
		IF Old_Shablon[i]<>0 AND New_Dinamo[i]=0 THEN
			shablonBufer[i]:=Old_Shablon[i];
		END_IF
				
	END_FOR
	Enable:= FALSE;
	
	//возвращаем получившийся (подкорректированный) шаблон
	Shablon:=shablonBufer;		
END_IF

END_FUNCTION_BLOCK

// Device/Application/Code/Modules_dinamogramma/Alarm_Control
// Контроль отклонений значений динамограммы
FUNCTION_BLOCK Alarm_Control
VAR_INPUT
	Shablon: ARRAY[0..500] OF REAL;
	Value: REAL;
	Index: INT;
	Otklonenie: REAL;
END_VAR
VAR_OUTPUT
	Alarm: BOOL;
	AlarmLogArr:ARRAY[0..500]OF AlarmLog;
END_VAR
VAR
	i_alarm:INT:=0;
	DTAlarm:DTime;
END_VAR

IF ABS(Shablon[Index]-Value) >= Otklonenie THEN
	Alarm:= TRUE;
	
	IF i_alarm>=500 THEN
		i_alarm:=0;
	END_IF
	
	AlarmLogArr[i_alarm].Date_Time:=plc_prg.DTime_0.sTimeStamp;
	AlarmLogArr[i_alarm].ShablonIndex:=Index;
	AlarmLogArr[i_alarm].ShablonValue:=Shablon[Index];
	AlarmLogArr[i_alarm].Value:=Value;
	AlarmLogArr[i_alarm].Otklonenie:=Otklonenie;
	
	i_alarm:=i_alarm+1;
	
	ELSE
		Alarm:=FALSE;
END_IF

END_FUNCTION_BLOCK

// Device/Application/Code/Modules_parameter/Emulate_Parameter_Power
FUNCTION_BLOCK Emulate_Parameter_Power
VAR_INPUT
	Enable:BOOL;
	U_Random_Min: INT;
	U_Random_Max: INT;
	I_Random_Min: INT;
	I_Random_Max: INT;
	Index: INT;
END_VAR
VAR_OUTPUT
	U:REAL;
	I:REAL;
	Work_Up: REAL;
	Work_Down: REAL;
	Work_Hod: REAL;
	Max_Power: REAL;
	Min_Power:REAL;
	Razmah: REAL;
END_VAR
VAR
	uBuffer: ARRAY[0..gvl.m_MAX_arr] OF REAL; //промежуточная переменная
	iBuffer: ARRAY[0..gvl.m_MAX_arr] OF REAL; //промежуточная переменная
	ind:INT;

END_VAR
VAR CONSTANT
	//m_MAX_arr: INT:=200; //размер массива	
	
END_VAR

IF Enable THEN	
	
	U:=OSCAT_BASIC.RDM2(last:=3 , low:=U_Random_Min , high:=U_Random_Max )*0.975;	//случайное значение напряжения
	I:=OSCAT_BASIC.RDM2(last:=7 , low:=I_Random_Min , high:=I_Random_Max )*0.948;	// случайное значение тока
	
	Index:=Index-1;
	
	uBuffer[Index]:=U;
	iBuffer[Index]:=I;
	
	
	
	IF Index=m_MAX_arr THEN
		FOR ind:=0 TO m_MAX_arr DO
				Work_Hod:=Work_Hod+uBuffer[Ind]*iBuffer[Ind]*0.1;	//работа за ход
			END_FOR
			Work_Hod:=Work_Hod/1000;
			
		FOR ind:=0 TO m_MAX_arr/2 DO
				Work_Up:=Work_Up+uBuffer[Ind]*iBuffer[Ind]*0.1;	//работа на подъеме
			END_FOR
			Work_Up:=Work_Up/1000;
			
		FOR ind:=m_MAX_arr/2 TO m_MAX_arr DO
				Work_Down:=Work_Down+uBuffer[Ind]*iBuffer[Ind]*0.1;	//работа на спуске
			END_FOR
			Work_Down:=Work_Down/1000;
		
		Max_Power:= MAX(uBuffer[0]*iBuffer[0], uBuffer[1]*iBuffer[1]);	
		Min_Power:= MIN(uBuffer[0]*iBuffer[0], uBuffer[1]*iBuffer[1]);	
		FOR ind:=2 TO m_MAX_arr DO
				Max_Power:=MAX(Max_Power, uBuffer[Ind]*iBuffer[Ind]);	//минимальная и максимальная мощность
				Min_Power:= MIN(Min_Power, uBuffer[Ind]*iBuffer[Ind]);
			END_FOR
			Max_Power:=Max_Power/1000;
			Min_Power:=Min_Power/1000;
		
			Razmah:= Max_Power - Min_Power;
	END_IF
	
	
	Enable:=FALSE;
END_IF

END_FUNCTION_BLOCK

// Device/Application/Code/Modules_parameter/Calculate_Parameter_Usilie
FUNCTION_BLOCK Calculate_Parameter_Usilie
VAR_INPUT
	Enable:BOOL;
	Index:INT;
	Dinamogramma: ARRAY[0..gvl.m_MAX_arr] OF REAL;
	
END_VAR
VAR_OUTPUT
	Work_Up: REAL;
	Work_Down: REAL;
	Work_Hod: REAL;
	Raznica: REAL;
	Max_Usil: REAL;
	Min_Usil:REAL;
	Razmah: REAL;
END_VAR
VAR
	ind:INT;
	DinaCount: INT;
	i:INT;
END_VAR
VAR CONSTANT
	//m_MAX_arr: INT:=200; //размер массива	
	
END_VAR

IF Enable THEN

	Index:=Index-1;

	Work_Up:=0;
	Work_Down:=0;
	Work_Hod:=0;
	WHILE Dinamogramma[i]<>0 AND Dinamogramma[i+1]<>0 AND Dinamogramma[i+1]<>0 DO
		i:=i+1;
	END_WHILE
	
	IF i>=gvl.m_MAX_arr THEN
		DinaCount:=gvl.m_MAX_arr;
	ELSE
		DinaCount:=i+1;
	END_IF
	
	
	//IF Index = DinaCount THEN
		
	FOR ind:=0 TO DinaCount DO
				Work_Hod:=Work_Hod+Dinamogramma[Ind];	//работа за ход
			END_FOR
	
	FOR ind:=0 TO DinaCount/2 DO
				Work_Up:=Work_Up+Dinamogramma[Ind];	//работа на подъеме
			END_FOR
			
		FOR ind:=DinaCount/2 TO DinaCount DO
				Work_Down:=Work_Down+Dinamogramma[Ind];	//работа на спуске
			END_FOR
			
		Raznica:= ABS(Work_Up - Work_Down);
		
		Max_Usil:= MAX(Dinamogramma[0], Dinamogramma[1]);	
		Min_Usil:= MIN(Dinamogramma[0], Dinamogramma[1]);	
		FOR ind:=2 TO DinaCount-1 DO
				Max_Usil:=MAX(Max_Usil, Dinamogramma[Ind]);	//минимальная и максимальная мощность
				Min_Usil:= MIN(Min_Usil, Dinamogramma[Ind]);
			END_FOR
		
			Razmah:= Max_Usil - Min_Usil;
	//END_IF

END_IF

END_FUNCTION_BLOCK

// Device/Application/Code/Dop_modules/NotNull
FUNCTION_BLOCK INTERNAL NotNull
VAR_INPUT
	Perem:WORD;
END_VAR
VAR_OUTPUT
	GoodPerem:WORD;
END_VAR
VAR
	NulLimit:INT;
END_VAR

IF Perem <> 0 THEN GoodPerem:=Perem; NulLimit:=0;
ELSE NulLimit:=NulLimit+1;
	IF NulLimit = 600 THEN 
		GoodPerem:=0; 
		NulLimit:=500;
	END_IF
END_IF

END_FUNCTION_BLOCK

// Device/Application/Code/Dop_modules/Perecl_Perem
FUNCTION_BLOCK Perecl_Perem
VAR_INPUT
	N: BYTE;
	VibrDvigZGor, VibrDvigZVert, VibrDvigZOs: REAL;
	VibrDvigPPElDvGor, VibrDvigPPElDvVert, VibrDvigPPElDvOs: REAL;
	VibrNasPGor, VibrNasPVert, VibrNasPOs: REAL;
	VibrNasZGor, VibrNasZVert, VibrNasZOs: REAL;
	Tok, DavlOut, DavlIn, Rashod, KPD, NagrevJidk, TempDvigZad, TempDvigPer, TempNasPer, TempNasZad: REAL;
END_VAR
VAR_OUTPUT
	Perem: REAL; 
END_VAR
VAR

	
END_VAR


	

IF Start=FALSE THEN 
	IF SaveConfig=TRUE THEN
		M1 := MemM1;
		M2 := MemM2;
		M3 := MemM3;
		M4 := MemM4;
		M5 := MemM5;
		M6 := MemM6;
		M7 := MemM7;
		M8 := MemM8;
		M9 := MemM9;
		M10 := MemM10;
		M11 := MemM11;
		M12 := MemM12;
		S1 := MemS1;
		S2 := MemS2;
		S3 := MemS3;
		S4 := MemS4;
		S5 := MemS5;
		S6 := MemS6;
		S7 := MemS7;
		S8 := MemS8;
		S9 := MemS9;
		S10 := MemS10;
		S11 := MemS11;
		S12 := MemS12;
	END_IF

	Start:=TRUE;
END_IF


VibrDvigZGor := ((VibrDvigZGor * M1 ) - S1);
VibrDvigZVert := ((VibrDvigZVert * M2) - S2);
VibrDvigZOs := ((VibrDvigZOs * M3) - S3);
VibrDvigPPElDvGor := ((VibrDvigPPElDvGor * M4) - S4);
VibrDvigPPElDvVert := ((VibrDvigPPElDvVert * M5) - S5);
VibrDvigPPElDvOs := ((VibrDvigPPElDvOs * M6) -S6);
VibrNasPGor := ((VibrNasPGor * M7) - S7);
VibrNasPVert := ((VibrNasPVert * M8) - S8);
VibrNasPOs := ((VibrNasPOs * M9) - S9);
VibrNasZGor := ((VibrNasZGor * M10) - S10);
VibrNasZVert := ((VibrNasZVert * M11) - S11);
VibrNasZOs := ((VibrNasZOs * M12) - S12);

IF VibrDvigZGor < 0 THEN VibrDvigZGor := 0; END_IF
IF VibrDvigZVert < 0 THEN VibrDvigZVert := 0; END_IF
IF VibrDvigZOs < 0 THEN VibrDvigZOs := 0; END_IF
IF VibrDvigPPElDvGor < 0 THEN VibrDvigPPElDvGor := 0; END_IF
IF VibrDvigPPElDvVert < 0 THEN VibrDvigPPElDvVert := 0; END_IF
IF VibrDvigPPElDvOs < 0 THEN VibrDvigPPElDvOs := 0; END_IF
IF VibrNasPGor < 0 THEN VibrNasPGor := 0; END_IF
IF VibrNasPVert < 0 THEN VibrNasPVert := 0; END_IF
IF VibrNasPOs < 0 THEN VibrNasPOs := 0; END_IF
IF VibrNasZGor < 0 THEN VibrNasZGor := 0; END_IF
IF VibrNasZVert < 0 THEN VibrNasZVert := 0; END_IF
IF VibrNasZOs < 0 THEN VibrNasZOs := 0; END_IF

VibrA1 := VibrDvigZGor;
VibrA2 := VibrDvigZVert;
VibrA3 := VibrDvigZOs;
VibrB1 := VibrDvigPPElDvGor;
VibrB2 := VibrDvigPPElDvVert;
VibrB3 := VibrDvigPPElDvOs;
VibrC1 := VibrNasPGor;
VibrC2 := VibrNasPVert;
VibrC3 := VibrNasPOs;
VibrD1 := VibrNasZGor;
VibrD2 := VibrNasZVert;
VibrD3 := VibrNasZOs;

IF N = 55 THEN Perem := VibrDvigZGor; ELSE
	IF N = 53 THEN Perem := VibrDvigZVert;ELSE
		IF N = 51 THEN Perem := VibrDvigZOs;ELSE
			IF N = 54 THEN Perem := VibrDvigPPElDvGor;ELSE
				IF N = 52 THEN Perem := VibrDvigPPElDvVert;ELSE
					IF N = 50 THEN Perem := VibrDvigPPElDvOs;ELSE
						IF N = 47 THEN Perem := VibrNasPGor;ELSE
							IF N = 45 THEN Perem := VibrNasPVert;ELSE
								IF N = 43 THEN Perem := VibrNasPOs;ELSE
									IF N = 46 THEN Perem := VibrNasZGor;ELSE
										IF N = 44 THEN Perem := VibrNasZVert;ELSE
											IF N = 42 THEN Perem := VibrNasZOs;ELSE
												IF N = 58 THEN Perem := Tok;ELSE
													IF N = 60 THEN Perem := DavlOut;ELSE
														IF N = 61 THEN Perem := DavlIn;ELSE
															IF N = 59 THEN Perem := Rashod;ELSE
																IF N = 56 THEN Perem := KPD;ELSE
																	IF N = 57 THEN Perem := NagrevJidk;ELSE
																		IF N = 49 THEN Perem := TempDvigZad;ELSE
																			IF N = 48 THEN Perem := TempDvigPer;ELSE
																				IF N = 41 THEN Perem := TempNasPer;ELSE
																					IF N = 40 THEN Perem := TempNasZad; 
																					END_IF
																				END_IF
																			END_IF
																		END_IF
																	END_IF
																END_IF
															END_IF
														END_IF
													END_IF
												END_IF
											END_IF
										END_IF
									END_IF
								END_IF
							END_IF
						END_IF
					END_IF
				END_IF
			END_IF
		END_IF
	END_IF
END_IF

END_FUNCTION_BLOCK

// Device/Application/Code/Dop_modules/Schetchik
FUNCTION_BLOCK Schetchik
VAR_INPUT
	On:BOOL;
	n_Start:BYTE;
	n_End:BYTE;
END_VAR
VAR_OUTPUT
	n_Actual:BYTE;
END_VAR
VAR
	n: BYTE := n_Start;
END_VAR

IF n>=n_End THEN n:=n_Start;
 ELSE
	IF On=TRUE THEN n:=n+1;
		n_Actual:=n;
	END_IF
END_IF

END_FUNCTION_BLOCK

// Device/Application/Code/Dop_modules/AddInMassive
FUNCTION_BLOCK AddInMassive
VAR_INPUT
	DateTime: STRING(20);
	Var1, Var2, Var3, Var4, Var5, Var6 : REAL;
END_VAR
VAR_OUTPUT
	Massiv:Massive;
END_VAR
VAR
END_VAR

Massiv.Date_Time:= DateTime;
Massiv.var1:=Var1;
Massiv.var2:=Var2;
Massiv.var3:=Var3;
Massiv.var4:=Var4;
Massiv.var5:=Var5;
Massiv.var6:=Var6;

END_FUNCTION_BLOCK

// Device/Application/Code/Dop_modules/convert
PROGRAM convert
VAR
	pt: POINTER TO WORD;
	W1: WORD;
	W2: WORD;
	perTest: WORD;
END_VAR

pt:=ADR(var2);
W1:=pt^;
pt:=pt+2;
W2:=pt^;
perTest:=458;

END_PROGRAM

// Device/Application/Code/Dop_modules/Duo_Word_to_Real
FUNCTION Duo_Word_to_Real : REAL
VAR_INPUT
	in1: WORD;
	in0: WORD;
END_VAR
VAR
	ptr: POINTER TO DWORD;
END_VAR

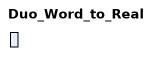
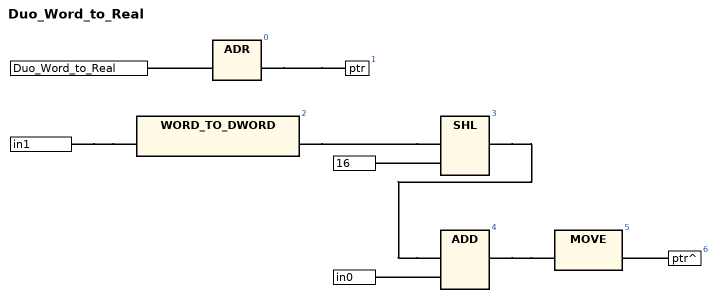
ptr := ADR(Duo_Word_to_Real);
ptr^ := SHL(WORD_TO_DWORD(in1), 16) + in0;

END_FUNCTION

// Device/Application/Code/Dop_modules/Real_to_Duo_Word
FUNCTION_BLOCK Real_to_Duo_Word
VAR_INPUT
	In: REAL;
END_VAR
VAR_OUTPUT
	Out_1 : WORD;
	Out_2 : WORD;
END_VAR
VAR
	pt: POINTER TO WORD;
END_VAR

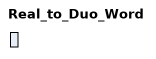
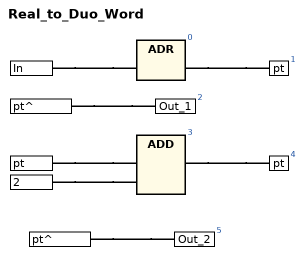
pt := ADR(In);
Out_1 := pt^;
pt := pt + 2;
Out_2 := pt^;

END_FUNCTION_BLOCK

// Device/Application/Code/Dop_modules/Timer_impuls
FUNCTION_BLOCK Timer_impuls
VAR_INPUT
	t: TIME;
END_VAR
VAR_OUTPUT
	Out_impuls: BOOL;
	Time_now: TIME;
END_VAR
VAR
	Timepulse: TP;
END_VAR
VAR // added by the converter: edge detectors and wires of the graphical bodies
    _w1 : ANY;
    _w2 : BOOL;
END_VAR

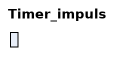
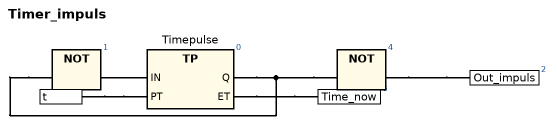
Timepulse(IN := _w1, PT := t); // TP
_w1 := NOT Timepulse.Q;
Out_impuls := _w2;
Time_now := Timepulse.ET;
_w2 := NOT Timepulse.Q;

END_FUNCTION_BLOCK

// Device/Application/Code/Dop_modules/IVD3_input_old
(*функциональный блок считывания состояния входов и код исключительных ситуаций модуля МВА8*)
FUNCTION_BLOCK IVD3_input_old
VAR_INPUT
	(*идентификатор порта*)								Handle:SysCom.RTS_IEC_HANDLE;
	(*разрешение на работу*)							Enabl:BOOL;
	(*режим работы ModBus, по умолчанию RTU*)			Modd:MB_MODE:=MB_RTU (*MB_RTU, MB_Ascii*);
	(*адресс прибора, по умолчанию 1*)					Addr:BYTE:=1;
	(*таймаут, по умолчанию 500мс*)						TimeOut: TIME:=T#500MS;(*таймаут*)
	(*число перезапросов, по умолчанию 3*)				ErCL:BYTE:=3;
END_VAR

VAR_OUTPUT
	(*измеренное значение 1го входа прибора*)			_z:REAL;
	(*измеренное значение 2го входа прибора*)			_x:REAL;
	(*измеренное значение 3го входа прибора*)			_y:REAL;
	
	(*код исключительной ситуации 1го канала*)			inpExcSCode1:WORD;
	(*код исключительной ситуации 2го канала*)			inpExcSCode2:WORD;
	(*код исключительной ситуации 3го канала*)			inpExcSCode3:WORD;

	(*код ошибки*)		wErrCode:WORD:=0;
	(*флаг завершения*)	done:BOOL:=FALSE;
END_VAR
VAR
	Err:WORD:=0;
	ErrCount:BYTE:=0;
	cmpl:BOOL;
	marker:WORD:=0;
	
	Exception: BYTE;
	DataSize: WORD;
	RegAddr1:WORD:=16#00;
	RegAddr2:WORD:=16#02;
	RegAddr3:WORD:=16#04;
	
	
	BUFFER: ARRAY [0..255] OF BYTE;
	x: REAL;
	ptr_x:POINTER TO BYTE;
	
		rtrig:R_TRIG;
	trig:rs;
	
	get_modbus: MB_RD_INP_REGS;
END_VAR

done:=FALSE;

rtrig(clk:=(Enabl));
trig(set:=rtrig.Q,RESET1:=FALSE);

CASE marker OF

0: get_modbus(
	Enable:=trig.Q1 ,			(* разрешение работы блока *)
	Mode:=Modd ,		(*режим передачи*)
	DevAddr:=Addr ,			(*адрес*)
	FirstAddr:=RegAddr1 ,			(*номер регистра*)
	Quantity:=6,			(*количество регистров*)
	ComHandle:=handle ,(*номер COM-порта*)
	TimeOut:=TimeOut , 		(*Таймаут T#50ms*)
	Buffer:=Buffer ,		(* буфер данных *)
	Complete=>cmpl ,		(* скопировать признак завершения операции *)
	Exception=>Err ,		(* скопировать регистр ошибок *)
	ByteCnt=>DataSize );		(*кол-во считанных байтов *)


IF cmpl THEN
	IF Err=0 THEN (*Если нет ошибок, то получаем данные из буфера типа INT*)
		x:=0;
		ptr_x:=ADR(x);
		
		ptr_x^:=buffer[4];
		ptr_x:=ptr_x+1;
		ptr_x^:=buffer[3];
		ptr_x:=ptr_x+1;
		ptr_x^:=buffer[6];
		ptr_x:=ptr_x+1;
		ptr_x^:=buffer[5];
		_z:=x;
		
		inpExcSCode1:=0;
		(*ptr_x:=ADR(inpExcSCode1);
		ptr_x^:=buffer[1];
		ptr_x:=ptr_x+1;
		ptr_x^:=buffer[0];*)
			
		
		marker:=1;
		ErrCount:=0;
		ELSE
			IF (ErrCount >= ErCL) THEN
				marker:=1;
				wErrCode:=Err;
				ErrCount:=0;
			END_IF
			ErrCount:=ErrCount+1;
	END_IF
END_IF

1:  get_modbus(
	Enable:=trig.Q1 ,			(* разрешение работы блока *)
	Mode:=Modd ,		(*режим передачи*)
	DevAddr:=Addr ,			(*адрес*)
	FirstAddr:=RegAddr2 ,			(*номер регистра*)
	Quantity:=2,			(*количество регистров*)
	ComHandle:=handle ,(*номер COM-порта*)
	TimeOut:=TimeOut , 		(*Таймаут T#50ms*)
	Buffer:=Buffer ,		(* буфер данных *)
	Complete=>cmpl ,		(* скопировать признак завершения операции *)
	Exception=>Err ,		(* скопировать регистр ошибок *)
	ByteCnt=>DataSize );		(*кол-во считанных байтов *)


IF cmpl THEN
	IF Err=0 THEN (*Если нет ошибок, то получаем данные из буфера типа INT*)
		x:=0;
		ptr_x:=ADR(x);
		ptr_x^:=buffer[4];
		ptr_x:=ptr_x+1;
		ptr_x^:=buffer[3];
		ptr_x:=ptr_x+1;
		ptr_x^:=buffer[6];
		ptr_x:=ptr_x+1;
		ptr_x^:=buffer[5];
		_x:=x;
		
		inpExcSCode2:=0;
		(*ptr_x:=ADR(inpExcSCode2);
		ptr_x^:=buffer[1];
		ptr_x:=ptr_x+1;
		ptr_x^:=buffer[0];*)
		
	
		marker:=2;
		ErrCount:=0;
		ELSE
			IF (ErrCount >= ErCL) THEN
				marker:=2;
				wErrCode:=Err;
				ErrCount:=0;
			END_IF
			ErrCount:=ErrCount+1;
	END_IF	
END_IF

2:  get_modbus(
	Enable:=trig.Q1 ,			(* разрешение работы блока *)
	Mode:=Modd ,		(*режим передачи*)
	DevAddr:=Addr ,			(*адрес*)
	FirstAddr:=RegAddr3 ,			(*номер регистра*)
	Quantity:=2,			(*количество регистров*)
	ComHandle:=handle ,(*номер COM-порта*)
	TimeOut:=TimeOut , 		(*Таймаут T#50ms*)
	Buffer:=Buffer ,		(* буфер данных *)
	Complete=>cmpl ,		(* скопировать признак завершения операции *)
	Exception=>Err ,		(* скопировать регистр ошибок *)
	ByteCnt=>DataSize );		(*кол-во считанных байтов *)


IF cmpl THEN
	IF Err=0 THEN (*Если нет ошибок, то получаем данные из буфера типа INT*)
		x:=0;
		ptr_x^:=buffer[4];
		ptr_x:=ptr_x+1;
		ptr_x^:=buffer[3];
		ptr_x:=ptr_x+1;
		ptr_x^:=buffer[6];
		ptr_x:=ptr_x+1;
		ptr_x^:=buffer[5];
		_y:=x;
	
		inpExcSCode3:=0;
		(*ptr_x:=ADR(inpExcSCode3);
		ptr_x^:=buffer[1];
		ptr_x:=ptr_x+1;
		ptr_x^:=buffer[0];*)
		
		
		marker:=0;
			done:=TRUE;
			trig(RESET1:=TRUE);
		ErrCount:=0;
		ELSE
			IF (ErrCount >= ErCL) THEN
				marker:=0;
				wErrCode:=Err;
				ErrCount:=0;
					done:=TRUE;
					trig(RESET1:=TRUE);
			END_IF
		ErrCount:=ErrCount+1;
	END_IF	
END_IF

END_CASE

END_FUNCTION_BLOCK

// Device/Application/Code/Dop_modules/POU
FUNCTION POU : string
VAR_INPUT
END_VAR
VAR
	GetSysDT:DTU.GetDateAndTime;    // ФБ cчитывания системного времени

	// считанное системное время:
	
	uiReadYear:			UINT;       // год
	uiReadMonth:		UINT;		// месяц
	uiReadDay:			UINT;       // день
	uiReadHour:			UINT;       // часы
	uiReadMinute:		UINT;       // минуты
	uiReadSecond:		UINT;       // секунды
	

	SetSysDT:DTU.SetDateAndTime;    // ФБ установки системного времени
	xWriteDT:			BOOL;       // триггер записи системного времени
	
	// устанавливаемое системное время
	
	uiWriteYear:		UINT:=2016; // год
	uiWriteMonth:		UINT:=1;    // месяц
	uiWriteDay:			UINT:=1;    // день
	uiWriteHour:		UINT;       // часы
	uiWriteMinute:		UINT;       // минуты
	uiWriteSecond:		UINT;       // секунды
	
	eWriteDTerror:		DTU.ERROR;  // статус работы функции DTConcat
END_VAR
VAR // added by the converter: edge detectors and wires of the graphical bodies
    _w1, _w2, _w3 : ANY;
END_VAR

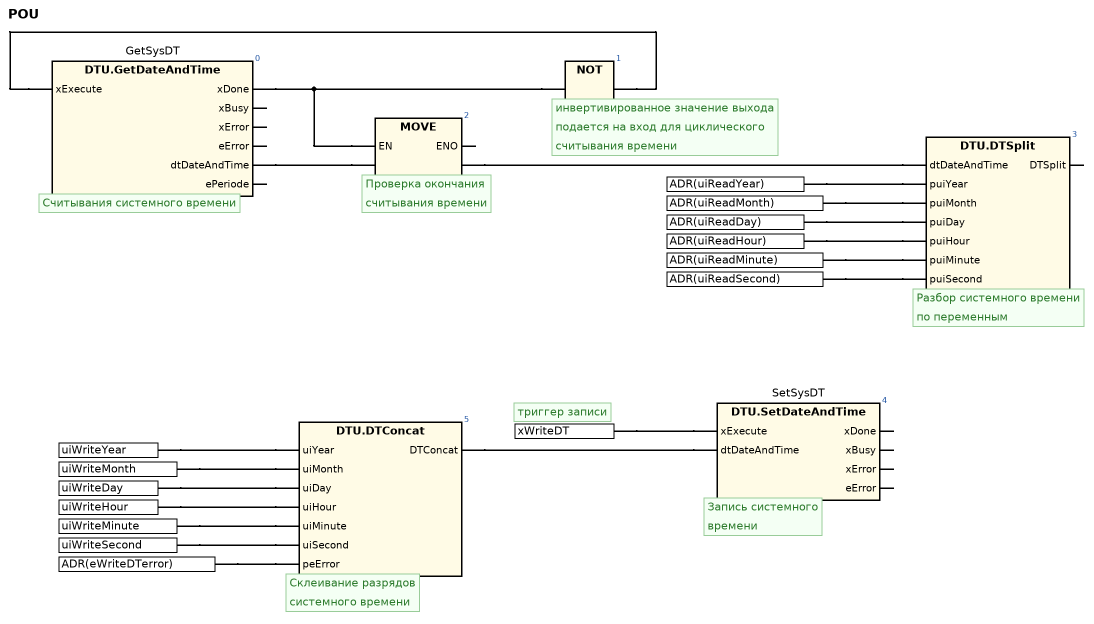
GetSysDT(xExecute := _w1); // DTU.GetDateAndTime
_w1 := NOT GetSysDT.xDone;
// инвертивированное значение выхода
// подается на вход для циклического
// считывания времени
// Проверка окончания
// считывания времени
IF GetSysDT.xDone THEN _w2 := GetSysDT.dtDateAndTime; END_IF
DTU.DTSplit(dtDateAndTime := _w2, puiYear := ADR(uiReadYear), puiMonth := ADR(uiReadMonth), puiDay := ADR(uiReadDay), puiHour := ADR(uiReadHour), puiMinute := ADR(uiReadMinute), puiSecond := ADR(uiReadSecond));
// Разбор системного времени
// по переменным
// Запись системного
// времени
SetSysDT(xExecute := xWriteDT, dtDateAndTime := _w3); // DTU.SetDateAndTime
// Cчитывания системного времени
// триггер записи
// Склеивание разрядов
// системного времени
_w3 := DTU.DTConcat(uiYear := uiWriteYear, uiMonth := uiWriteMonth, uiDay := uiWriteDay, uiHour := uiWriteHour, uiMinute := uiWriteMinute, uiSecond := uiWriteSecond, peError := ADR(eWriteDTerror));

END_FUNCTION

// Device/Application/Code/Modules_dinamogramma/Create_Shablon
// Формирование шаблона динамограммы с использованием некоторого количеаства проходов
FUNCTION_BLOCK Create_Shablon
VAR_INPUT
	Prohod: INT;
	Value: REAL;
	Index: INT;
	Size_dinamo:INT;
END_VAR
VAR_OUTPUT
	State: BOOL;
	Shablon: ARRAY[0..500] OF REAL;
END_VAR
VAR
	shablonBufer: ARRAY[0..500] OF REAL;
	prohod_i:INT:=1;
	i:INT;
END_VAR

IF State=FALSE THEN
	// Если количество проходов еще не истекло, то выполняем сбор данных
	IF Prohod >= prohod_i THEN
		shablonBufer[Index]:= shablonBufer[Index]+Value;
		IF Index = Size_dinamo THEN
			prohod_i:= prohod_i + 1;
		END_IF
		
		
	// Если получены все массивы, делим на кол-во проходов и получаем среднее значение
	IF Prohod = prohod_i THEN
			FOR i:=0 TO Size_dinamo DO
				shablonBufer[i]:= shablonBufer[i]/Prohod;
			END_FOR
			State:= TRUE;	// Выставляем флаг о завершернии в TRUE
			Shablon:= shablonBufer; 	// Предоставляем полученный усредненный массив
		END_IF 
	END_IF
END_IF

END_FUNCTION_BLOCK

// Device/Application/Code/Modules/SMS
FUNCTION_BLOCK SMS
VAR_INPUT
END_VAR
VAR_OUTPUT
END_VAR
VAR
	ComConn_sms: ComConn;
END_VAR

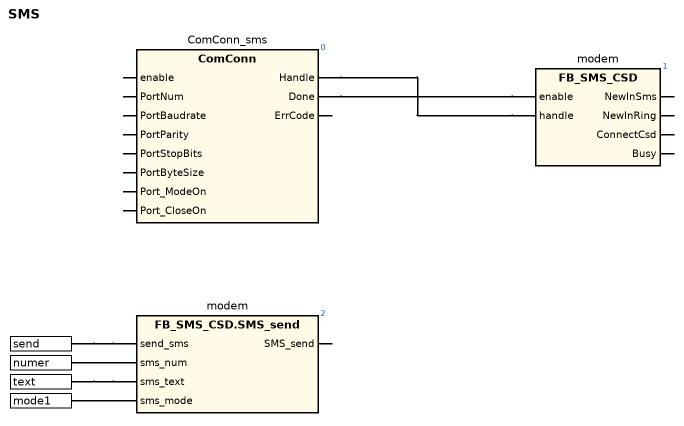
ComConn_sms(); // ComConn
modem(enable := ComConn_sms.Done, handle := ComConn_sms.Handle); // FB_SMS_CSD
modem.SMS_send(send_sms := send, sms_num := numer, sms_text := text, sms_mode := mode1);

END_FUNCTION_BLOCK

// Device/Application/Code/Dop_modules/IVD3_input
FUNCTION_BLOCK IVD3_input_reg_123
VAR_INPUT
	(*идентификатор порта*)											Handle:SysCom.RTS_IEC_HANDLE;
	(*разрешение на работу*)										Enabl:BOOL;
	(*адресс прибора, по умолчанию 1*)								Addr:BYTE:=1;
	(*таймаут, по умолчанию 30мс*)									TimeOut: TIME:=T#30MS;
	
	TextTimeNow: STRING;
	LengthMassive:INT;

END_VAR
VAR_OUTPUT
	(*измеренное значение плоскости X*)			X:REAL;
	(*измеренное значение плоскости Y*)			Y:REAL;
	(*измеренное значение плоскости Z*)			Z:REAL;
	
	cmpl:BOOL;
	valRecd:bool;
	iCompl:UINT;
	(*код ошибки*)										wErrCode:WORD;
	(*флаг завершения*)									done:BOOL;
END_VAR
VAR
	(*режим работы ModBus (MB_RTU, MB_Ascii), по умолчанию RTU*)	Modd:MB_MODE:=MB_RTU ;
	(*адресс регистра, по умолчанию 0*)								RegAddr:WORD:=16#0;
	(*число перезапросов, по умолчанию 3*)							ErCL:BYTE:=3;
	ErrCount:BYTE:=0;
	
	shag:byte:=0;
	err:WORD;
	Exception: BYTE;
	DataSize: WORD;
	KolReg:BYTE;
	get_modbus:MB_RD_INP_REGS;
	//get_modbus2:MB_RD_INP_REGS;
	BUFFER: ARRAY [0..255] OF BYTE;
	i: WORD;
	
	_x, _y, _z: REAL;
	ptr_x, ptr_y, ptr_z:POINTER TO BYTE;
	
	rtrig:R_TRIG;
	trig:rs;
END_VAR

done:=FALSE;
valRecd:=FALSE;

rtrig(clk:=(Enabl));
trig(set:=rtrig.Q,RESET1:=FALSE);


get_modbus(
	Enable:=trig.Q1 ,			(* разрешение работы блока *)
	Mode:=Modd ,		(*режим передачи*)
	DevAddr:=Addr ,			(*адрес*)
	FirstAddr:=RegAddr ,			(*номер регистра*)
	Quantity:=6,			(*количество регистров*)
	ComHandle:=Handle ,(*номер COM-порта*)
	TimeOut:=TimeOut , 		(*Таймаут T#30ms*)
	Buffer:=Buffer ,		(* буфер данных *)
	Complete=>cmpl ,		(* скопировать признак завершения операции *)
	Exception=>Err ,		(* скопировать регистр ошибок *)
	ByteCnt=>DataSize );		(*кол-во считанных байтов *)

//IF cmpl=TRUE THEN
//	IF iCompl>=65500 THEN
//		iCompl:=0;
//	END_IF
//	iCompl:=iCompl+1;
//END_IF


	//IF cmpl THEN
		IF Err=0 THEN	
			IF DataSize=17 THEN
//cmpl:=FALSE;
		_z:=0;
		ptr_z:=ADR(z);
		ptr_z^:=buffer[4];
		ptr_z:=ptr_z+1;
		ptr_z^:=buffer[3];
		ptr_z:=ptr_z+1;
		ptr_z^:=buffer[6];
		ptr_z:=ptr_z+1;
		ptr_z^:=buffer[5];
		Z:=_z;
		
		_x:=0;
		ptr_x:=ADR(x);
		ptr_x^:=buffer[8];
		ptr_x:=ptr_x+1;
		ptr_x^:=buffer[7];
		ptr_x:=ptr_x+1;
		ptr_x^:=buffer[10];
		ptr_x:=ptr_x+1;
		ptr_x^:=buffer[9];
		X:=_x;
		
		_y:=0;
		ptr_y:=ADR(y);
		ptr_y^:=buffer[12];
		ptr_y:=ptr_y+1;
		ptr_y^:=buffer[11];
		ptr_y:=ptr_y+1;
		ptr_y^:=buffer[14];
		ptr_y:=ptr_y+1;
		ptr_y^:=buffer[13];
		Y:=_y;
			
		valRecd:= true;

		done:=TRUE;
		trig(RESET1:=TRUE);
		ErrCount:=0;
		wErrCode:=Err;
		IF iCompl>=65500 THEN
			iCompl:=0;
		END_IF
	iCompl:=iCompl+1;
	ELSE
	ErrCount:=ErrCount+1;
		IF (ErrCount >= ErCL) THEN
			ErrCount:=0;
			done:=TRUE;
			trig(RESET1:=TRUE);
			wErrCode:=Err;
		END_IF
	END_IF
END_IF

//END_IF

END_FUNCTION_BLOCK

// Device/Application/Code/Modules_dinamogramma/Auton_dynamogram_modbus
FUNCTION_BLOCK Auton_dynamogram_modbus
VAR_INPUT
	(*идентификатор порта*)													Handle:SysCom.RTS_IEC_HANDLE;
	(*разрешение на работу*)													Enabl:BOOL;
	(*адресс прибора, по умолчанию 1*)								Addr:BYTE:=30;
	(*таймаут, по умолчанию 30мс*)										TimeOut: TIME:=T#30MS;
	//(*размер массива динамограммы, по умолчанию 250*)	Length: INT:=250;
END_VAR
VAR_OUTPUT
	(*Динамограмма*)																Dynamogram: ARRAY[0..gvl.Dynamogram_length] OF INT;
	(*Статус получения ответа после запроса*)					cmpl:BOOL;
	(*флаг завершения*)															done: BOOL;
	valRecd:BOOL;
	(*Просто счётчик для просмотра работы*)						iCompl:UINT;
END_VAR
VAR
	(*режим работы ModBus (MB_RTU, MB_Ascii), по умолчанию RTU*)		Modd:MB_MODE:=MB_RTU ;
	(*адресс регистра, по умолчанию 0*)												RegAddr:WORD:=16#F0;
	(*число перезапросов, по умолчанию 3*)										ErCL:BYTE:=3;
	(*Объект для отправки запросов и получения ответов по протоколу modbus*)	get_modbus:MB_RD_HOLD_REGS;
	(*Буфер для принятых байт ответа*)												BUFFER: ARRAY [0..255] OF BYTE;
	
	(*Количество ошибок*)																		ErrCount:BYTE:=0;
	(*Регистр ошибок*)																				err:WORD;
	(*Количество считанных байт*)															DataSize: WORD;
	
	(*Значение из ответа*)																		_value:INT;
	(*Указатель переменной*) 																ptr_value:POINTER TO BYTE;
	(*Собранное значение*) 																	Value:INT;
	
	(*Переключатель состояний (true/false) *)											rtrig:R_TRIG;
	(*Переключатель состояний (true/false)*)											trig:rs;
	
	i:INT:=0;
	
END_VAR

done:=FALSE;
valRecd:=FALSE;
i:=0;
//WHILE i<=gvl.Dynamogram_length DO
FOR i:=0 TO gvl.Dynamogram_length DO
	valRecd


	
rtrig(clk:=(Enabl));
trig(set:=rtrig.Q, RESET1:=FALSE);



	

get_modbus(
	Enable:=trig.Q1 ,				(* разрешение работы блока *)
	Mode:=Modd ,					(*режим передачи*)
	DevAddr:=Addr ,				(*адрес*)
	FirstAddr:=RegAddr ,		(*номер регистра*)
	Quantity:=1,						(*количество регистров*)
	ComHandle:=handle ,		(*номер COM-порта*)
	TimeOut:=TimeOut , 		(*Таймаут T#30ms*)
	Buffer:=Buffer ,					(* буфер данных *)
	Complete=>cmpl ,			(* скопировать признак завершения операции *)
	Exception=>Err ,				(* скопировать регистр ошибок *)
	ByteCnt=>DataSize );		(*кол-во считанных байтов *)
	

	
IF cmpl AND Err=0 THEN	
	IF DataSize=7 THEN
		value:=0;
		ptr_value:=ADR(value);
		ptr_value^:=buffer[4];
		ptr_value:=ptr_value+1;
		ptr_value^:=buffer[3];
		Value:=value;		
			
		valRecd:= true;

		
		trig(RESET1:=TRUE);
		ErrCount:=0;
		//wErrCode:=Err;
		IF iCompl>=65500 THEN
			iCompl:=0;
		END_IF
	iCompl:=iCompl+1;
	ELSE
	ErrCount:=ErrCount+1;
		IF (ErrCount >= ErCL) THEN
			ErrCount:=0;
			done:=TRUE;
			trig(RESET1:=TRUE);
			//wErrCode:=Err;
		END_IF
	END_IF
		
END_IF
Enabl:=TRUE;
IF cmpl=TRUE AND valRecd=TRUE THEN
	Dynamogram[i]:=Value;
	i:=i+1;
END_IF

//END_WHILE
END_FOR
Enabl:=FALSE;
done:=TRUE;

END_FUNCTION_BLOCK
